PROGRAM P2_03_Production_Ctrl
VAR
	bFeeding_Active						:BOOL;
	bMixing_Active						:BOOL;
	bDischarging_Active					:BOOL;
	
	bDischargeCloseRequest				:BOOL;
	bDischargeOpenRequest				:BOOL;
END_VAR
VAR // added by the converter: edge detectors and wires of the graphical bodies
    _w1, _w2, _w3 : BOOL;
END_VAR

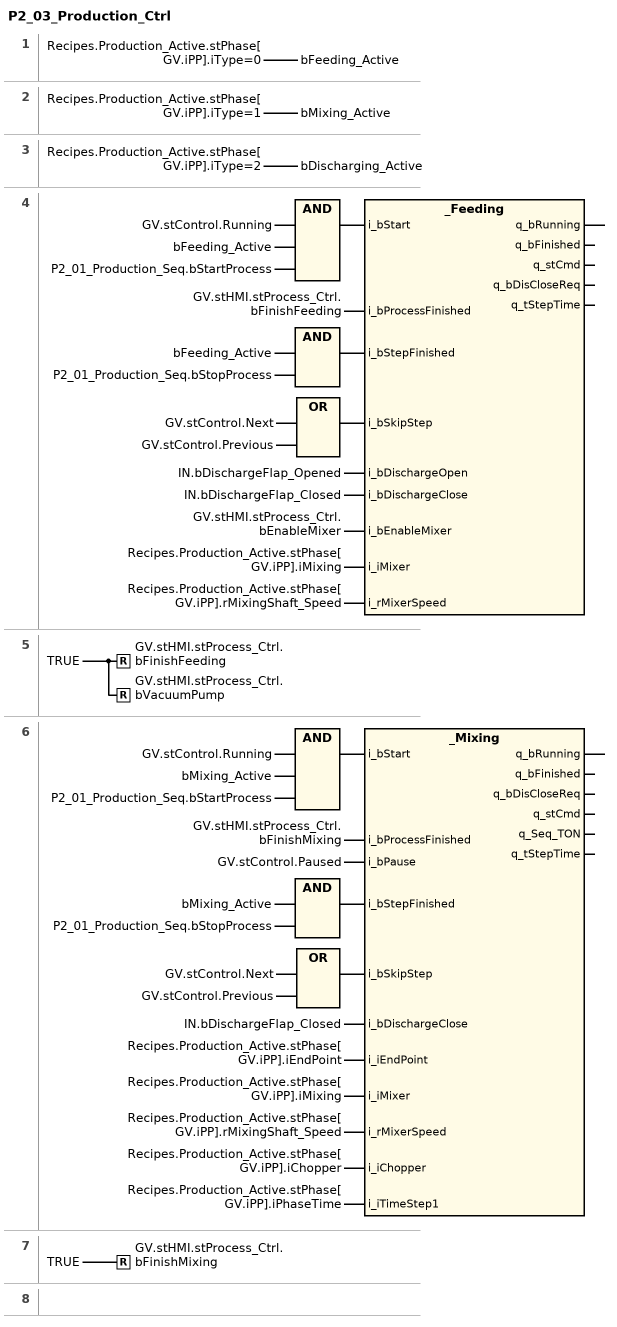
// NETWORK 1
bFeeding_Active := Recipes.Production_Active.stPhase[GV.iPP].iType=0;

// NETWORK 2
bMixing_Active := Recipes.Production_Active.stPhase[GV.iPP].iType=1;

// NETWORK 3
bDischarging_Active := Recipes.Production_Active.stPhase[GV.iPP].iType=2;

// NETWORK 4
_Feeding(i_bStart := GV.stControl.Running AND bFeeding_Active AND P2_01_Production_Seq.bStartProcess, i_bProcessFinished := GV.stHMI.stProcess_Ctrl.bFinishFeeding, i_bStepFinished := bFeeding_Active AND P2_01_Production_Seq.bStopProcess, i_bSkipStep := GV.stControl.Next OR GV.stControl.Previous, i_bDischargeOpen := IN.bDischargeFlap_Opened, i_bDischargeClose := IN.bDischargeFlap_Closed, i_bEnableMixer := GV.stHMI.stProcess_Ctrl.bEnableMixer, i_iMixer := Recipes.Production_Active.stPhase[GV.iPP].iMixing, i_rMixerSpeed := Recipes.Production_Active.stPhase[GV.iPP].rMixingShaft_Speed);

// NETWORK 5
GV.stHMI.stProcess_Ctrl.bFinishFeeding R= TRUE;
GV.stHMI.stProcess_Ctrl.bVacuumPump R= TRUE;

// NETWORK 6
_Mixing(i_bStart := GV.stControl.Running AND bMixing_Active AND P2_01_Production_Seq.bStartProcess, i_bProcessFinished := GV.stHMI.stProcess_Ctrl.bFinishMixing, i_bPause := GV.stControl.Paused, i_bStepFinished := bMixing_Active AND P2_01_Production_Seq.bStopProcess, i_bSkipStep := GV.stControl.Next OR GV.stControl.Previous, i_bDischargeClose := IN.bDischargeFlap_Closed, i_iEndPoint := Recipes.Production_Active.stPhase[GV.iPP].iEndPoint, i_iMixer := Recipes.Production_Active.stPhase[GV.iPP].iMixing, i_rMixerSpeed := Recipes.Production_Active.stPhase[GV.iPP].rMixingShaft_Speed, i_iChopper := Recipes.Production_Active.stPhase[GV.iPP].iChopper, i_iTimeStep1 := Recipes.Production_Active.stPhase[GV.iPP].iPhaseTime);

// NETWORK 7
GV.stHMI.stProcess_Ctrl.bFinishMixing R= TRUE;

// NETWORK 8

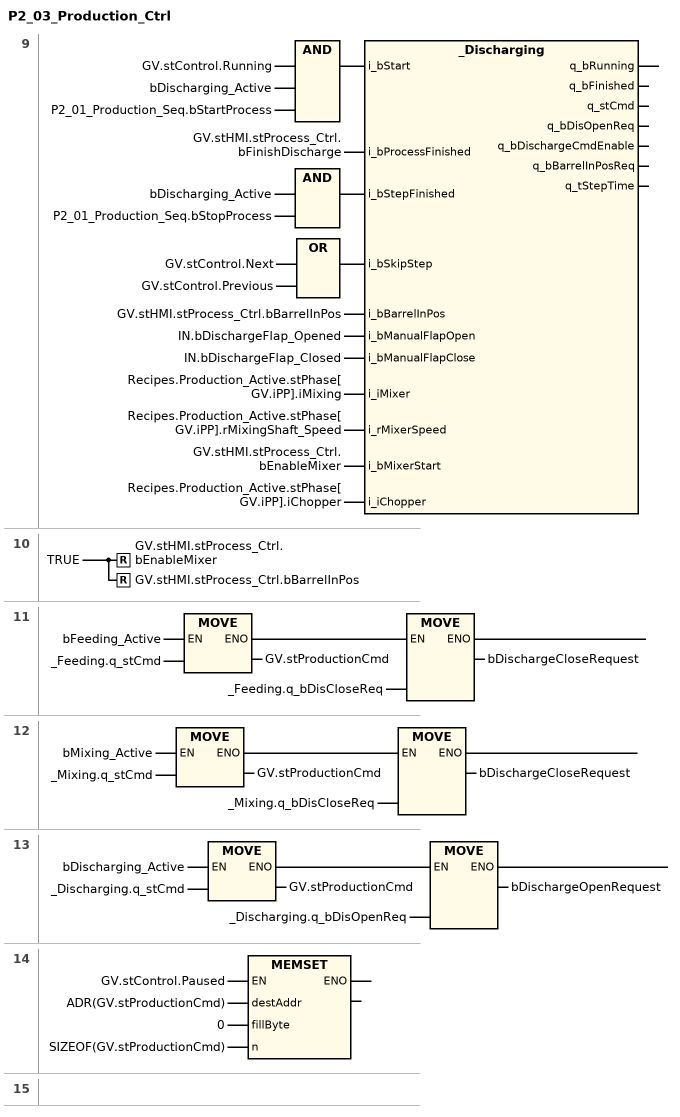
// NETWORK 9
_Discharging(i_bStart := GV.stControl.Running AND bDischarging_Active AND P2_01_Production_Seq.bStartProcess, i_bProcessFinished := GV.stHMI.stProcess_Ctrl.bFinishDischarge, i_bStepFinished := bDischarging_Active AND P2_01_Production_Seq.bStopProcess, i_bSkipStep := GV.stControl.Next OR GV.stControl.Previous, i_bBarrelInPos := GV.stHMI.stProcess_Ctrl.bBarrelInPos, i_bManualFlapOpen := IN.bDischargeFlap_Opened, i_bManualFlapClose := IN.bDischargeFlap_Closed, i_iMixer := Recipes.Production_Active.stPhase[GV.iPP].iMixing, i_rMixerSpeed := Recipes.Production_Active.stPhase[GV.iPP].rMixingShaft_Speed, i_bMixerStart := GV.stHMI.stProcess_Ctrl.bEnableMixer, i_iChopper := Recipes.Production_Active.stPhase[GV.iPP].iChopper);

// NETWORK 10
GV.stHMI.stProcess_Ctrl.bEnableMixer R= TRUE;
GV.stHMI.stProcess_Ctrl.bBarrelInPos R= TRUE;

// NETWORK 11
_w1 := bFeeding_Active;
IF _w1 THEN GV.stProductionCmd := _Feeding.q_stCmd; END_IF
IF _w1 THEN bDischargeCloseRequest := _Feeding.q_bDisCloseReq; END_IF

// NETWORK 12
_w2 := bMixing_Active;
IF _w2 THEN GV.stProductionCmd := _Mixing.q_stCmd; END_IF
IF _w2 THEN bDischargeCloseRequest := _Mixing.q_bDisCloseReq; END_IF

// NETWORK 13
_w3 := bDischarging_Active;
IF _w3 THEN GV.stProductionCmd := _Discharging.q_stCmd; END_IF
IF _w3 THEN bDischargeOpenRequest := _Discharging.q_bDisOpenReq; END_IF

// NETWORK 14
IF GV.stControl.Paused THEN
    MEMSET(destAddr := ADR(GV.stProductionCmd), fillByte := 0, n := SIZEOF(GV.stProductionCmd));
END_IF

// NETWORK 15

END_PROGRAM

(* stored: Version 1.1.0.1
   POU P2_03_Production_Ctrl: Id {583d7fc6-053b-4f96-9a94-d52b256ea881}, SpecialFunc None *)
